// Mitsubishi GX Developer project: PLC_PCO520L2   PLC: Q06UDEH   Autoclave Auto Flow

PROGRAM AT_AC
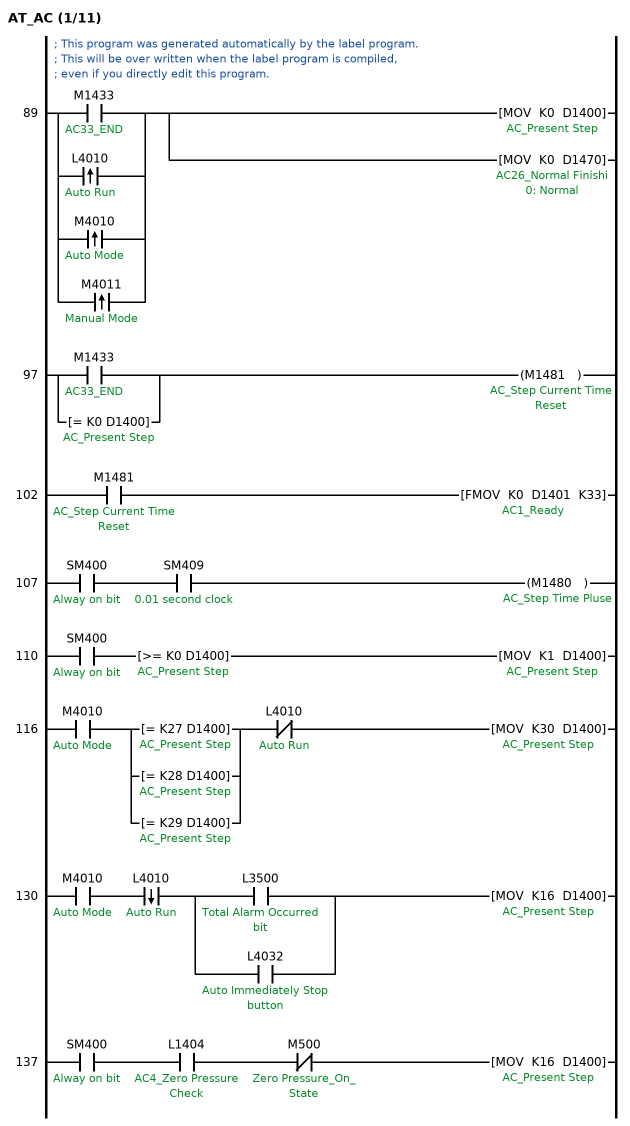
; This program was generated automatically by the label program.
; This will be over written when the label program is compiled,
; even if you directly edit this program.
89    LD      M1433  ; AC33_END
      ORP     L4010  ; Auto Run
      ORP     M4010  ; Auto Mode
      ORP     M4011  ; Manual Mode
      MOV     K0 D1400  ; AC_Present Step
      MOV     K0 D1470  ; AC26_Normal Finishi 0: Normal
97    LD      M1433  ; AC33_END
      OR=     K0 D1400  ; AC_Present Step
      OUT     M1481  ; AC_Step Current Time Reset
102   LD      M1481  ; AC_Step Current Time Reset
      FMOV    K0 D1401 K33  ; AC1_Ready
107   LD      SM400  ; Alway on bit
      AND     SM409  ; 0.01 second clock
      OUT     M1480  ; AC_Step Time Pluse
110   LD      SM400  ; Alway on bit
      AND>=   K0 D1400  ; AC_Present Step
      MOV     K1 D1400
116   LD      M4010  ; Auto Mode
      LD=     K27 D1400  ; AC_Present Step
      OR=     K28 D1400  ; AC_Present Step
      OR=     K29 D1400  ; AC_Present Step
      ANB
      ANI     L4010  ; Auto Run
      MOV     K30 D1400
130   LD      M4010  ; Auto Mode
      ANDF    L4010  ; Auto Run
      LD      L3500  ; Total Alarm Occurred bit
      OR      L4032  ; Auto Immediately Stop button
      ANB
      MOV     K16 D1400
137   LD      SM400  ; Alway on bit
      AND     L1404  ; AC4_Zero Pressure Check
      ANI     M500  ; Zero Pressure_On_State
      MOV     K16 D1400
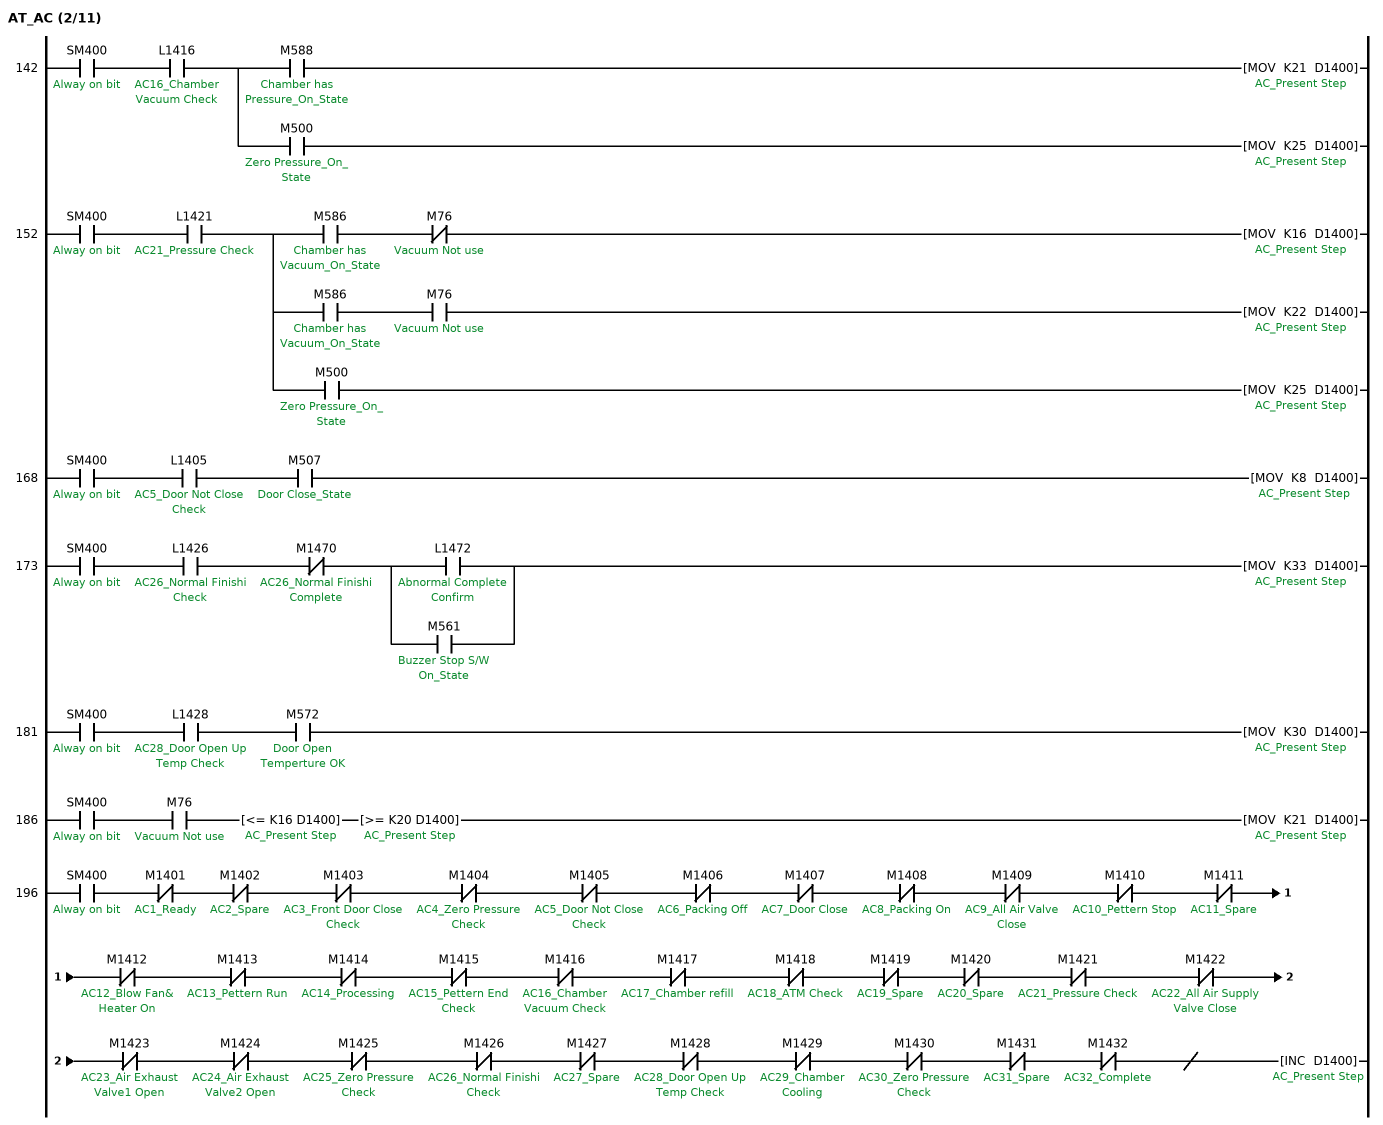
142   LD      SM400  ; Alway on bit
      AND     L1416  ; AC16_Chamber Vacuum Check
      MPS
      AND     M588  ; Chamber has Pressure_On_State
      MOV     K21 D1400
      MPP
      AND     M500  ; Zero Pressure_On_State
      MOV     K25 D1400
152   LD      SM400  ; Alway on bit
      AND     L1421  ; AC21_Pressure Check
      MPS
      AND     M586  ; Chamber has Vacuum_On_State
      ANI     M76  ; Vacuum Not use
      MOV     K16 D1400
      MRD
      AND     M586  ; Chamber has Vacuum_On_State
      AND     M76  ; Vacuum Not use
      MOV     K22 D1400
      MPP
      AND     M500  ; Zero Pressure_On_State
      MOV     K25 D1400
168   LD      SM400  ; Alway on bit
      AND     L1405  ; AC5_Door Not Close Check
      AND     M507  ; Door Close_State
      MOV     K8 D1400
173   LD      SM400  ; Alway on bit
      AND     L1426  ; AC26_Normal Finishi Check
      ANI     M1470  ; AC26_Normal Finishi Complete
      LD      L1472  ; Abnormal Complete Confirm
      OR      M561  ; Buzzer Stop S/W On_State
      ANB
      MOV     K33 D1400
181   LD      SM400  ; Alway on bit
      AND     L1428  ; AC28_Door Open Up Temp Check
      AND     M572  ; Door Open Temperture OK
      MOV     K30 D1400
186   LD      SM400  ; Alway on bit
      AND     M76  ; Vacuum Not use
      AND<=   K16 D1400  ; AC_Present Step
      AND>=   K20 D1400  ; AC_Present Step
      MOV     K21 D1400
196   LD      SM400  ; Alway on bit
      ANI     M1401  ; AC1_Ready
      ANI     M1402  ; AC2_Spare
      ANI     M1403  ; AC3_Front Door Close Check
      ANI     M1404  ; AC4_Zero Pressure Check
      ANI     M1405  ; AC5_Door Not Close Check
      ANI     M1406  ; AC6_Packing Off
      ANI     M1407  ; AC7_Door Close
      ANI     M1408  ; AC8_Packing On
      ANI     M1409  ; AC9_All Air Valve Close
      ANI     M1410  ; AC10_Pettern Stop
      ANI     M1411  ; AC11_Spare
      ANI     M1412  ; AC12_Blow Fan& Heater On
      ANI     M1413  ; AC13_Pettern Run
      ANI     M1414  ; AC14_Processing
      ANI     M1415  ; AC15_Pettern End Check
      ANI     M1416  ; AC16_Chamber Vacuum Check
      ANI     M1417  ; AC17_Chamber refill
      ANI     M1418  ; AC18_ATM Check
      ANI     M1419  ; AC19_Spare
      ANI     M1420  ; AC20_Spare
      ANI     M1421  ; AC21_Pressure Check
      ANI     M1422  ; AC22_All Air Supply Valve Close
      ANI     M1423  ; AC23_Air Exhaust Valve1 Open
      ANI     M1424  ; AC24_Air Exhaust Valve2 Open
      ANI     M1425  ; AC25_Zero Pressure Check
      ANI     M1426  ; AC26_Normal Finishi Check
      ANI     M1427  ; AC27_Spare
      ANI     M1428  ; AC28_Door Open Up Temp Check
      ANI     M1429  ; AC29_Chamber Cooling
      ANI     M1430  ; AC30_Zero Pressure Check
      ANI     M1431  ; AC31_Spare
      ANI     M1432  ; AC32_Complete
      INV
      INC     D1400
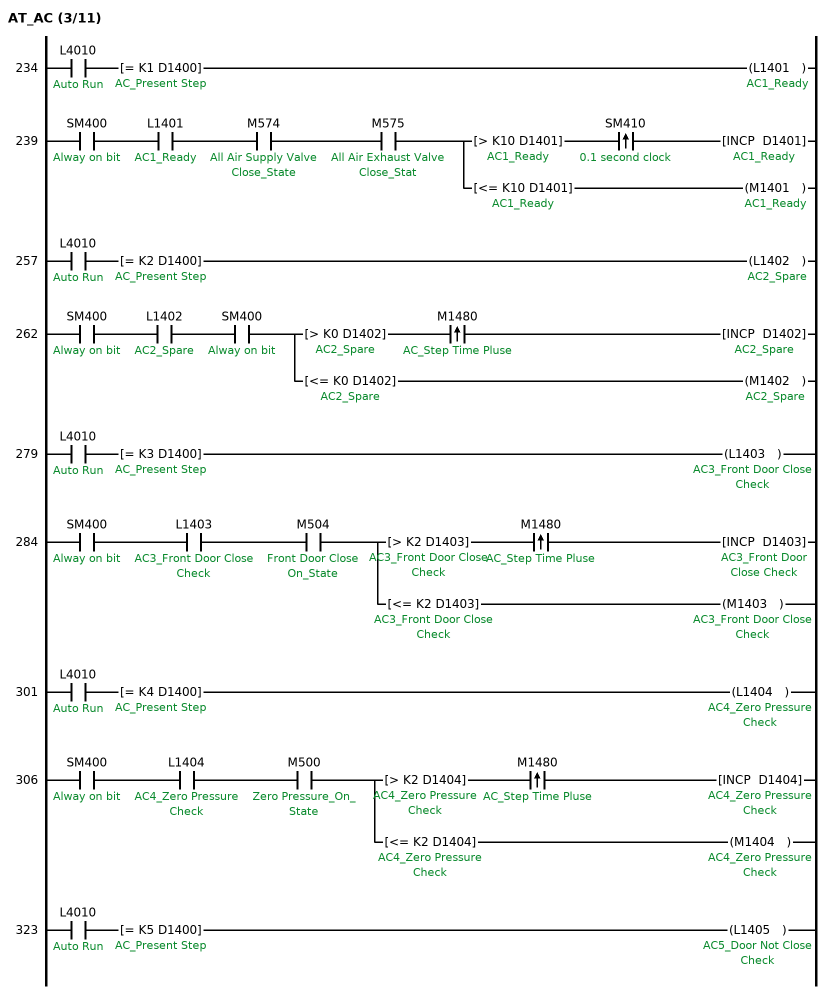
; 
234   LD      L4010  ; Auto Run
      AND=    K1 D1400  ; AC_Present Step
      OUT     L1401  ; AC1_Ready
239   LD      SM400  ; Alway on bit
      AND     L1401  ; AC1_Ready
      AND     M574  ; All Air Supply Valve Close_State
      AND     M575  ; All Air Exhaust Valve Close_Stat
      MPS
      AND>    K10 D1401  ; AC1_Ready
      ANDP    SM410  ; 0.1 second clock
      INCP    D1401
      MPP
      AND<=   K10 D1401  ; AC1_Ready
      OUT     M1401  ; AC1_Ready
; 
257   LD      L4010  ; Auto Run
      AND=    K2 D1400  ; AC_Present Step
      OUT     L1402  ; AC2_Spare
262   LD      SM400  ; Alway on bit
      AND     L1402  ; AC2_Spare
      AND     SM400  ; Alway on bit
      MPS
      AND>    K0 D1402  ; AC2_Spare
      ANDP    M1480  ; AC_Step Time Pluse
      INCP    D1402
      MPP
      AND<=   K0 D1402  ; AC2_Spare
      OUT     M1402  ; AC2_Spare
; 
279   LD      L4010  ; Auto Run
      AND=    K3 D1400  ; AC_Present Step
      OUT     L1403  ; AC3_Front Door Close Check
284   LD      SM400  ; Alway on bit
      AND     L1403  ; AC3_Front Door Close Check
      AND     M504  ; Front Door Close On_State
      MPS
      AND>    K2 D1403  ; AC3_Front Door Close Check
      ANDP    M1480  ; AC_Step Time Pluse
      INCP    D1403
      MPP
      AND<=   K2 D1403  ; AC3_Front Door Close Check
      OUT     M1403  ; AC3_Front Door Close Check
; 
301   LD      L4010  ; Auto Run
      AND=    K4 D1400  ; AC_Present Step
      OUT     L1404  ; AC4_Zero Pressure Check
306   LD      SM400  ; Alway on bit
      AND     L1404  ; AC4_Zero Pressure Check
      AND     M500  ; Zero Pressure_On_State
      MPS
      AND>    K2 D1404  ; AC4_Zero Pressure Check
      ANDP    M1480  ; AC_Step Time Pluse
      INCP    D1404
      MPP
      AND<=   K2 D1404  ; AC4_Zero Pressure Check
      OUT     M1404  ; AC4_Zero Pressure Check
; 
323   LD      L4010  ; Auto Run
      AND=    K5 D1400  ; AC_Present Step
      OUT     L1405  ; AC5_Door Not Close Check
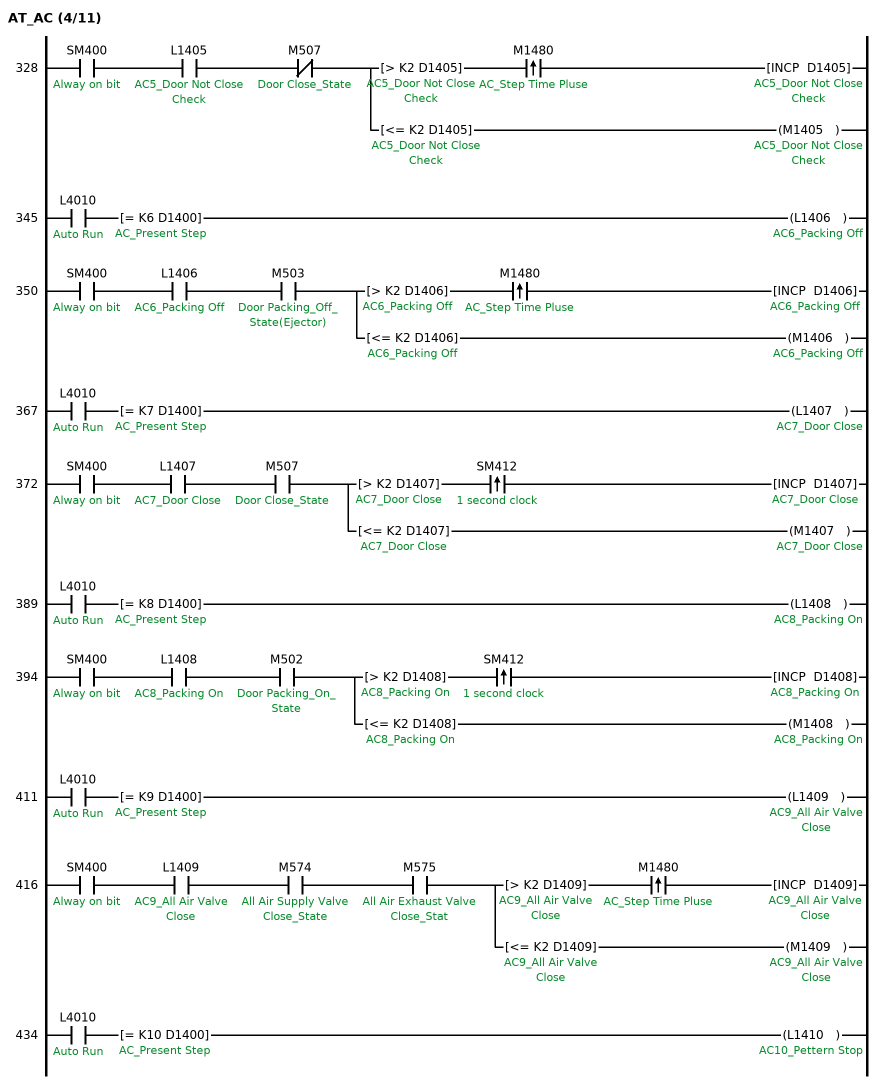
328   LD      SM400  ; Alway on bit
      AND     L1405  ; AC5_Door Not Close Check
      ANI     M507  ; Door Close_State
      MPS
      AND>    K2 D1405  ; AC5_Door Not Close Check
      ANDP    M1480  ; AC_Step Time Pluse
      INCP    D1405
      MPP
      AND<=   K2 D1405  ; AC5_Door Not Close Check
      OUT     M1405  ; AC5_Door Not Close Check
; 
345   LD      L4010  ; Auto Run
      AND=    K6 D1400  ; AC_Present Step
      OUT     L1406  ; AC6_Packing Off
350   LD      SM400  ; Alway on bit
      AND     L1406  ; AC6_Packing Off
      AND     M503  ; Door Packing_Off_State(Ejector)
      MPS
      AND>    K2 D1406  ; AC6_Packing Off
      ANDP    M1480  ; AC_Step Time Pluse
      INCP    D1406
      MPP
      AND<=   K2 D1406  ; AC6_Packing Off
      OUT     M1406  ; AC6_Packing Off
; 
367   LD      L4010  ; Auto Run
      AND=    K7 D1400  ; AC_Present Step
      OUT     L1407  ; AC7_Door Close
372   LD      SM400  ; Alway on bit
      AND     L1407  ; AC7_Door Close
      AND     M507  ; Door Close_State
      MPS
      AND>    K2 D1407  ; AC7_Door Close
      ANDP    SM412  ; 1 second clock
      INCP    D1407
      MPP
      AND<=   K2 D1407  ; AC7_Door Close
      OUT     M1407  ; AC7_Door Close
; 
389   LD      L4010  ; Auto Run
      AND=    K8 D1400  ; AC_Present Step
      OUT     L1408  ; AC8_Packing On
394   LD      SM400  ; Alway on bit
      AND     L1408  ; AC8_Packing On
      AND     M502  ; Door Packing_On_State
      MPS
      AND>    K2 D1408  ; AC8_Packing On
      ANDP    SM412  ; 1 second clock
      INCP    D1408
      MPP
      AND<=   K2 D1408  ; AC8_Packing On
      OUT     M1408  ; AC8_Packing On
; 
411   LD      L4010  ; Auto Run
      AND=    K9 D1400  ; AC_Present Step
      OUT     L1409  ; AC9_All Air Valve Close
416   LD      SM400  ; Alway on bit
      AND     L1409  ; AC9_All Air Valve Close
      AND     M574  ; All Air Supply Valve Close_State
      AND     M575  ; All Air Exhaust Valve Close_Stat
      MPS
      AND>    K2 D1409  ; AC9_All Air Valve Close
      ANDP    M1480  ; AC_Step Time Pluse
      INCP    D1409
      MPP
      AND<=   K2 D1409  ; AC9_All Air Valve Close
      OUT     M1409  ; AC9_All Air Valve Close
; 
434   LD      L4010  ; Auto Run
      AND=    K10 D1400  ; AC_Present Step
      OUT     L1410  ; AC10_Pettern Stop
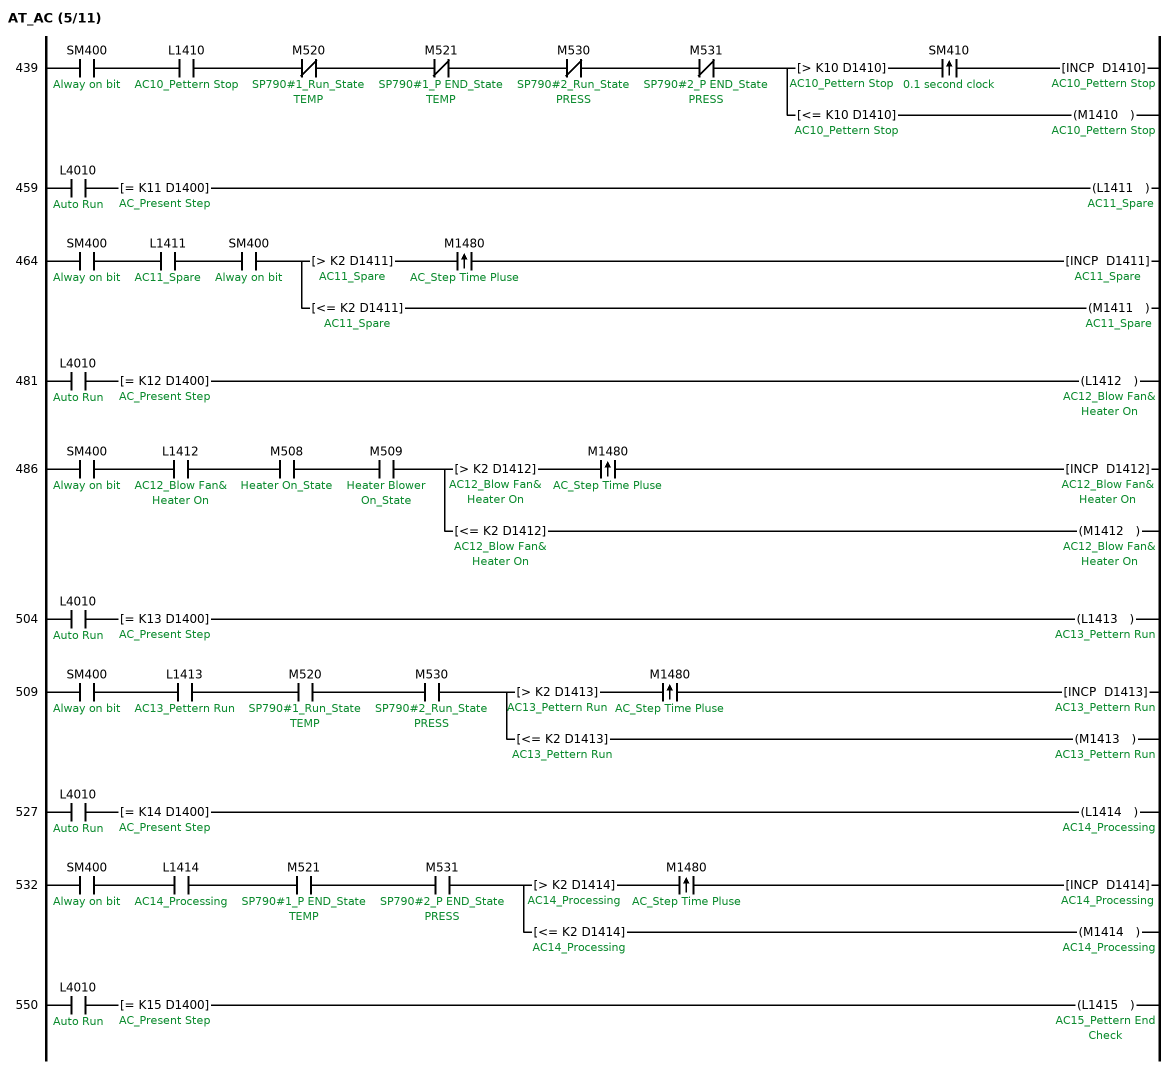
439   LD      SM400  ; Alway on bit
      AND     L1410  ; AC10_Pettern Stop
      ANI     M520  ; SP790#1_Run_State TEMP
      ANI     M521  ; SP790#1_P END_State TEMP
      ANI     M530  ; SP790#2_Run_State PRESS
      ANI     M531  ; SP790#2_P END_State PRESS
      MPS
      AND>    K10 D1410  ; AC10_Pettern Stop
      ANDP    SM410  ; 0.1 second clock
      INCP    D1410
      MPP
      AND<=   K10 D1410  ; AC10_Pettern Stop
      OUT     M1410  ; AC10_Pettern Stop
; 
459   LD      L4010  ; Auto Run
      AND=    K11 D1400  ; AC_Present Step
      OUT     L1411  ; AC11_Spare
464   LD      SM400  ; Alway on bit
      AND     L1411  ; AC11_Spare
      AND     SM400  ; Alway on bit
      MPS
      AND>    K2 D1411  ; AC11_Spare
      ANDP    M1480  ; AC_Step Time Pluse
      INCP    D1411
      MPP
      AND<=   K2 D1411  ; AC11_Spare
      OUT     M1411  ; AC11_Spare
; 
481   LD      L4010  ; Auto Run
      AND=    K12 D1400  ; AC_Present Step
      OUT     L1412  ; AC12_Blow Fan& Heater On
486   LD      SM400  ; Alway on bit
      AND     L1412  ; AC12_Blow Fan& Heater On
      AND     M508  ; Heater On_State
      AND     M509  ; Heater Blower On_State
      MPS
      AND>    K2 D1412  ; AC12_Blow Fan& Heater On
      ANDP    M1480  ; AC_Step Time Pluse
      INCP    D1412
      MPP
      AND<=   K2 D1412  ; AC12_Blow Fan& Heater On
      OUT     M1412  ; AC12_Blow Fan& Heater On
; 
504   LD      L4010  ; Auto Run
      AND=    K13 D1400  ; AC_Present Step
      OUT     L1413  ; AC13_Pettern Run
509   LD      SM400  ; Alway on bit
      AND     L1413  ; AC13_Pettern Run
      AND     M520  ; SP790#1_Run_State TEMP
      AND     M530  ; SP790#2_Run_State PRESS
      MPS
      AND>    K2 D1413  ; AC13_Pettern Run
      ANDP    M1480  ; AC_Step Time Pluse
      INCP    D1413
      MPP
      AND<=   K2 D1413  ; AC13_Pettern Run
      OUT     M1413  ; AC13_Pettern Run
; 
527   LD      L4010  ; Auto Run
      AND=    K14 D1400  ; AC_Present Step
      OUT     L1414  ; AC14_Processing
532   LD      SM400  ; Alway on bit
      AND     L1414  ; AC14_Processing
      AND     M521  ; SP790#1_P END_State TEMP
      AND     M531  ; SP790#2_P END_State PRESS
      MPS
      AND>    K2 D1414  ; AC14_Processing
      ANDP    M1480  ; AC_Step Time Pluse
      INCP    D1414
      MPP
      AND<=   K2 D1414  ; AC14_Processing
      OUT     M1414  ; AC14_Processing
; 
550   LD      L4010  ; Auto Run
      AND=    K15 D1400  ; AC_Present Step
      OUT     L1415  ; AC15_Pettern End Check
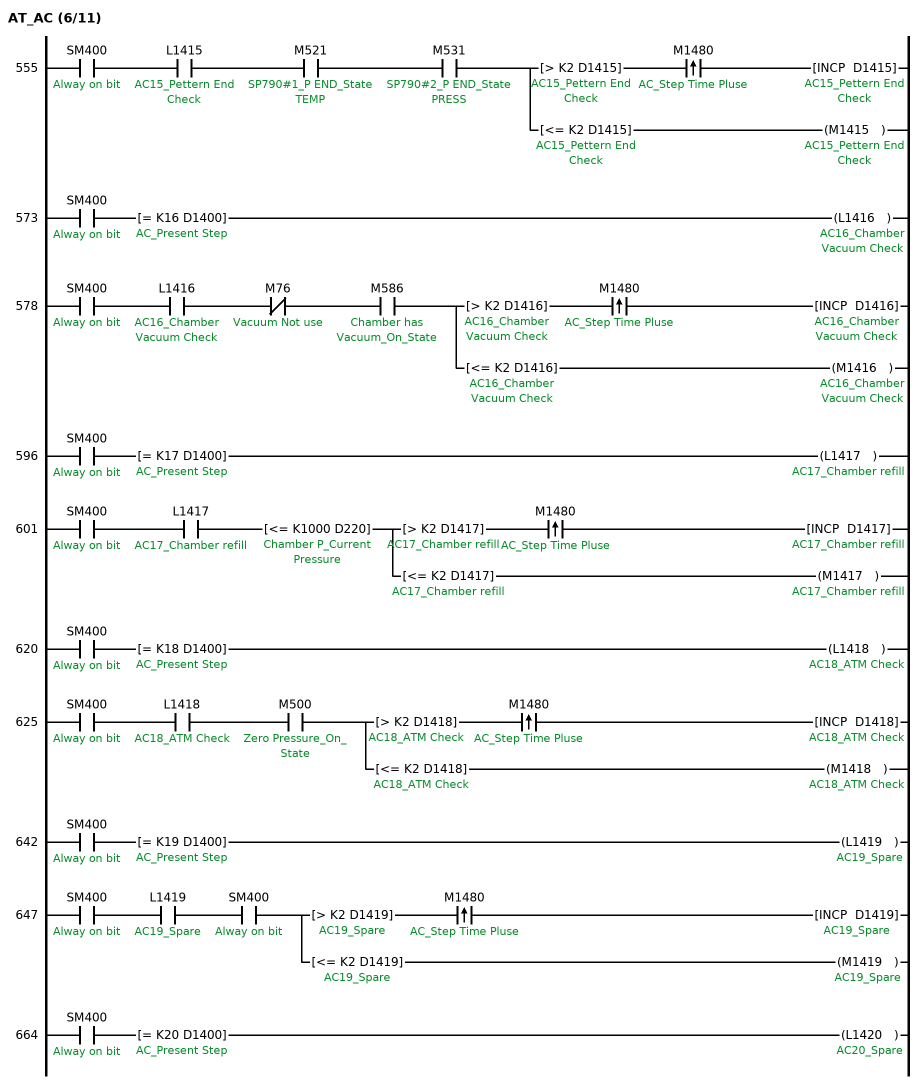
555   LD      SM400  ; Alway on bit
      AND     L1415  ; AC15_Pettern End Check
      AND     M521  ; SP790#1_P END_State TEMP
      AND     M531  ; SP790#2_P END_State PRESS
      MPS
      AND>    K2 D1415  ; AC15_Pettern End Check
      ANDP    M1480  ; AC_Step Time Pluse
      INCP    D1415
      MPP
      AND<=   K2 D1415  ; AC15_Pettern End Check
      OUT     M1415  ; AC15_Pettern End Check
; 
573   LD      SM400  ; Alway on bit
      AND=    K16 D1400  ; AC_Present Step
      OUT     L1416  ; AC16_Chamber Vacuum Check
578   LD      SM400  ; Alway on bit
      AND     L1416  ; AC16_Chamber Vacuum Check
      ANI     M76  ; Vacuum Not use
      AND     M586  ; Chamber has Vacuum_On_State
      MPS
      AND>    K2 D1416  ; AC16_Chamber Vacuum Check
      ANDP    M1480  ; AC_Step Time Pluse
      INCP    D1416
      MPP
      AND<=   K2 D1416  ; AC16_Chamber Vacuum Check
      OUT     M1416  ; AC16_Chamber Vacuum Check
; 
596   LD      SM400  ; Alway on bit
      AND=    K17 D1400  ; AC_Present Step
      OUT     L1417  ; AC17_Chamber refill
601   LD      SM400  ; Alway on bit
      AND     L1417  ; AC17_Chamber refill
      AND<=   K1000 D220  ; Chamber P_Current Pressure
      MPS
      AND>    K2 D1417  ; AC17_Chamber refill
      ANDP    M1480  ; AC_Step Time Pluse
      INCP    D1417
      MPP
      AND<=   K2 D1417  ; AC17_Chamber refill
      OUT     M1417  ; AC17_Chamber refill
; 
620   LD      SM400  ; Alway on bit
      AND=    K18 D1400  ; AC_Present Step
      OUT     L1418  ; AC18_ATM Check
625   LD      SM400  ; Alway on bit
      AND     L1418  ; AC18_ATM Check
      AND     M500  ; Zero Pressure_On_State
      MPS
      AND>    K2 D1418  ; AC18_ATM Check
      ANDP    M1480  ; AC_Step Time Pluse
      INCP    D1418
      MPP
      AND<=   K2 D1418  ; AC18_ATM Check
      OUT     M1418  ; AC18_ATM Check
; 
642   LD      SM400  ; Alway on bit
      AND=    K19 D1400  ; AC_Present Step
      OUT     L1419  ; AC19_Spare
647   LD      SM400  ; Alway on bit
      AND     L1419  ; AC19_Spare
      AND     SM400  ; Alway on bit
      MPS
      AND>    K2 D1419  ; AC19_Spare
      ANDP    M1480  ; AC_Step Time Pluse
      INCP    D1419
      MPP
      AND<=   K2 D1419  ; AC19_Spare
      OUT     M1419  ; AC19_Spare
; 
664   LD      SM400  ; Alway on bit
      AND=    K20 D1400  ; AC_Present Step
      OUT     L1420  ; AC20_Spare
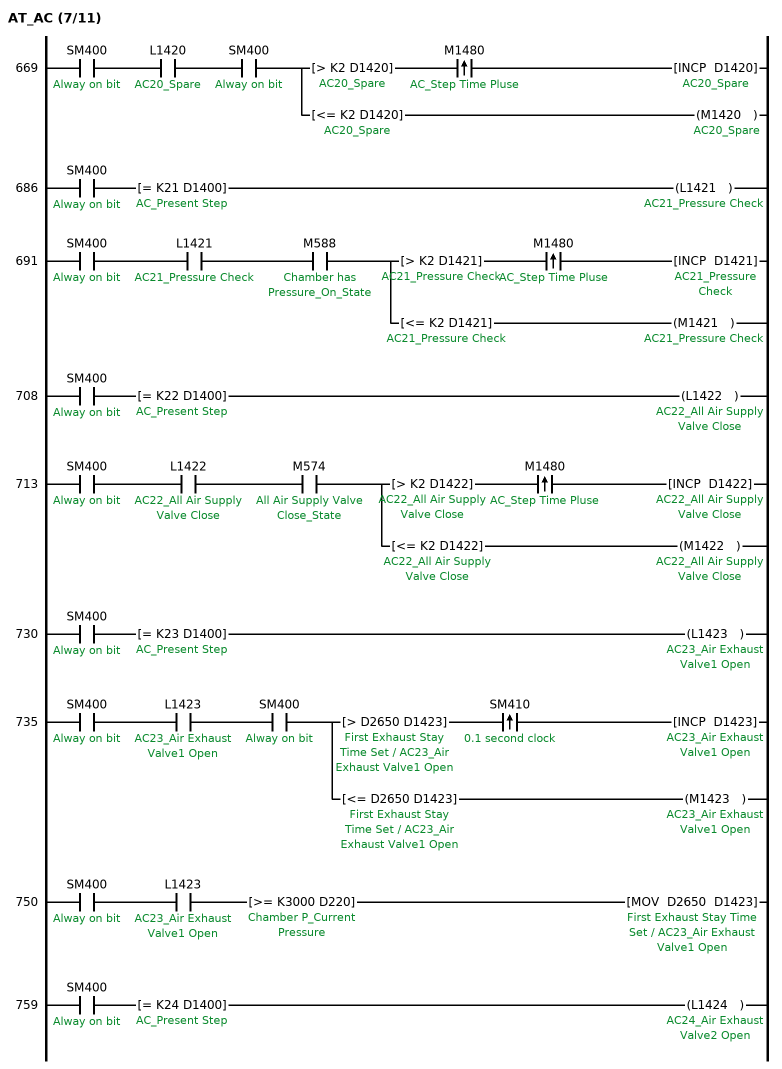
669   LD      SM400  ; Alway on bit
      AND     L1420  ; AC20_Spare
      AND     SM400  ; Alway on bit
      MPS
      AND>    K2 D1420  ; AC20_Spare
      ANDP    M1480  ; AC_Step Time Pluse
      INCP    D1420
      MPP
      AND<=   K2 D1420  ; AC20_Spare
      OUT     M1420  ; AC20_Spare
; 
686   LD      SM400  ; Alway on bit
      AND=    K21 D1400  ; AC_Present Step
      OUT     L1421  ; AC21_Pressure Check
691   LD      SM400  ; Alway on bit
      AND     L1421  ; AC21_Pressure Check
      AND     M588  ; Chamber has Pressure_On_State
      MPS
      AND>    K2 D1421  ; AC21_Pressure Check
      ANDP    M1480  ; AC_Step Time Pluse
      INCP    D1421
      MPP
      AND<=   K2 D1421  ; AC21_Pressure Check
      OUT     M1421  ; AC21_Pressure Check
; 
708   LD      SM400  ; Alway on bit
      AND=    K22 D1400  ; AC_Present Step
      OUT     L1422  ; AC22_All Air Supply Valve Close
713   LD      SM400  ; Alway on bit
      AND     L1422  ; AC22_All Air Supply Valve Close
      AND     M574  ; All Air Supply Valve Close_State
      MPS
      AND>    K2 D1422  ; AC22_All Air Supply Valve Close
      ANDP    M1480  ; AC_Step Time Pluse
      INCP    D1422
      MPP
      AND<=   K2 D1422  ; AC22_All Air Supply Valve Close
      OUT     M1422  ; AC22_All Air Supply Valve Close
; 
730   LD      SM400  ; Alway on bit
      AND=    K23 D1400  ; AC_Present Step
      OUT     L1423  ; AC23_Air Exhaust Valve1 Open
735   LD      SM400  ; Alway on bit
      AND     L1423  ; AC23_Air Exhaust Valve1 Open
      AND     SM400  ; Alway on bit
      MPS
      AND>    D2650 D1423  ; First Exhaust Stay Time Set / AC23_Air Exhaust Valve1 Open
      ANDP    SM410  ; 0.1 second clock
      INCP    D1423
      MPP
      AND<=   D2650 D1423  ; First Exhaust Stay Time Set / AC23_Air Exhaust Valve1 Open
      OUT     M1423  ; AC23_Air Exhaust Valve1 Open
750   LD      SM400  ; Alway on bit
      AND     L1423  ; AC23_Air Exhaust Valve1 Open
      AND>=   K3000 D220  ; Chamber P_Current Pressure
      MOV     D2650 D1423
; 
759   LD      SM400  ; Alway on bit
      AND=    K24 D1400  ; AC_Present Step
      OUT     L1424  ; AC24_Air Exhaust Valve2 Open
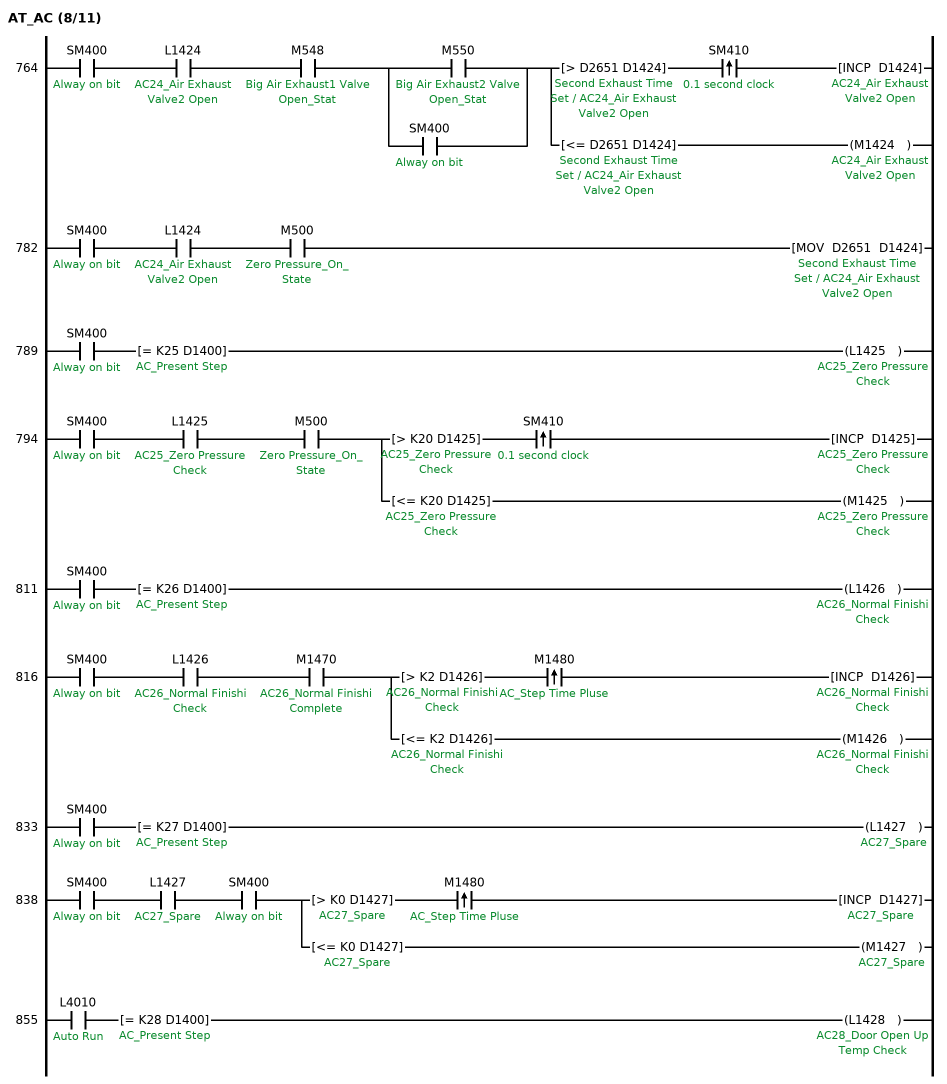
764   LD      SM400  ; Alway on bit
      AND     L1424  ; AC24_Air Exhaust Valve2 Open
      AND     M548  ; Big Air Exhaust1 Valve Open_Stat
      LD      M550  ; Big Air Exhaust2 Valve Open_Stat
      OR      SM400  ; Alway on bit
      ANB
      MPS
      AND>    D2651 D1424  ; Second Exhaust Time Set / AC24_Air Exhaust Valve2 Open
      ANDP    SM410  ; 0.1 second clock
      INCP    D1424
      MPP
      AND<=   D2651 D1424  ; Second Exhaust Time Set / AC24_Air Exhaust Valve2 Open
      OUT     M1424  ; AC24_Air Exhaust Valve2 Open
782   LD      SM400  ; Alway on bit
      AND     L1424  ; AC24_Air Exhaust Valve2 Open
      AND     M500  ; Zero Pressure_On_State
      MOV     D2651 D1424
; 
789   LD      SM400  ; Alway on bit
      AND=    K25 D1400  ; AC_Present Step
      OUT     L1425  ; AC25_Zero Pressure Check
794   LD      SM400  ; Alway on bit
      AND     L1425  ; AC25_Zero Pressure Check
      AND     M500  ; Zero Pressure_On_State
      MPS
      AND>    K20 D1425  ; AC25_Zero Pressure Check
      ANDP    SM410  ; 0.1 second clock
      INCP    D1425
      MPP
      AND<=   K20 D1425  ; AC25_Zero Pressure Check
      OUT     M1425  ; AC25_Zero Pressure Check
; 
811   LD      SM400  ; Alway on bit
      AND=    K26 D1400  ; AC_Present Step
      OUT     L1426  ; AC26_Normal Finishi Check
816   LD      SM400  ; Alway on bit
      AND     L1426  ; AC26_Normal Finishi Check
      AND     M1470  ; AC26_Normal Finishi Complete
      MPS
      AND>    K2 D1426  ; AC26_Normal Finishi Check
      ANDP    M1480  ; AC_Step Time Pluse
      INCP    D1426
      MPP
      AND<=   K2 D1426  ; AC26_Normal Finishi Check
      OUT     M1426  ; AC26_Normal Finishi Check
; 
833   LD      SM400  ; Alway on bit
      AND=    K27 D1400  ; AC_Present Step
      OUT     L1427  ; AC27_Spare
838   LD      SM400  ; Alway on bit
      AND     L1427  ; AC27_Spare
      AND     SM400  ; Alway on bit
      MPS
      AND>    K0 D1427  ; AC27_Spare
      ANDP    M1480  ; AC_Step Time Pluse
      INCP    D1427
      MPP
      AND<=   K0 D1427  ; AC27_Spare
      OUT     M1427  ; AC27_Spare
; 
855   LD      L4010  ; Auto Run
      AND=    K28 D1400  ; AC_Present Step
      OUT     L1428  ; AC28_Door Open Up Temp Check
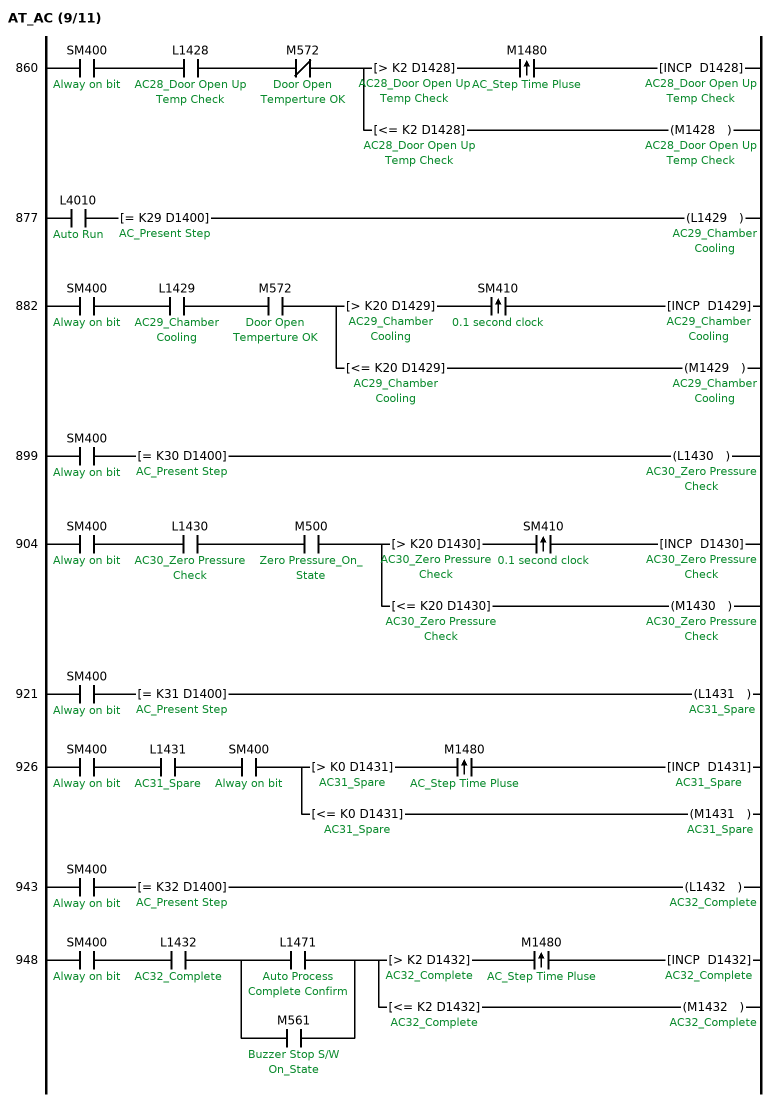
860   LD      SM400  ; Alway on bit
      AND     L1428  ; AC28_Door Open Up Temp Check
      ANI     M572  ; Door Open Temperture OK
      MPS
      AND>    K2 D1428  ; AC28_Door Open Up Temp Check
      ANDP    M1480  ; AC_Step Time Pluse
      INCP    D1428
      MPP
      AND<=   K2 D1428  ; AC28_Door Open Up Temp Check
      OUT     M1428  ; AC28_Door Open Up Temp Check
; 
877   LD      L4010  ; Auto Run
      AND=    K29 D1400  ; AC_Present Step
      OUT     L1429  ; AC29_Chamber Cooling
882   LD      SM400  ; Alway on bit
      AND     L1429  ; AC29_Chamber Cooling
      AND     M572  ; Door Open Temperture OK
      MPS
      AND>    K20 D1429  ; AC29_Chamber Cooling
      ANDP    SM410  ; 0.1 second clock
      INCP    D1429
      MPP
      AND<=   K20 D1429  ; AC29_Chamber Cooling
      OUT     M1429  ; AC29_Chamber Cooling
; 
899   LD      SM400  ; Alway on bit
      AND=    K30 D1400  ; AC_Present Step
      OUT     L1430  ; AC30_Zero Pressure Check
904   LD      SM400  ; Alway on bit
      AND     L1430  ; AC30_Zero Pressure Check
      AND     M500  ; Zero Pressure_On_State
      MPS
      AND>    K20 D1430  ; AC30_Zero Pressure Check
      ANDP    SM410  ; 0.1 second clock
      INCP    D1430
      MPP
      AND<=   K20 D1430  ; AC30_Zero Pressure Check
      OUT     M1430  ; AC30_Zero Pressure Check
; 
921   LD      SM400  ; Alway on bit
      AND=    K31 D1400  ; AC_Present Step
      OUT     L1431  ; AC31_Spare
926   LD      SM400  ; Alway on bit
      AND     L1431  ; AC31_Spare
      AND     SM400  ; Alway on bit
      MPS
      AND>    K0 D1431  ; AC31_Spare
      ANDP    M1480  ; AC_Step Time Pluse
      INCP    D1431
      MPP
      AND<=   K0 D1431  ; AC31_Spare
      OUT     M1431  ; AC31_Spare
; 
943   LD      SM400  ; Alway on bit
      AND=    K32 D1400  ; AC_Present Step
      OUT     L1432  ; AC32_Complete
948   LD      SM400  ; Alway on bit
      AND     L1432  ; AC32_Complete
      LD      L1471  ; Auto Process Complete Confirm
      OR      M561  ; Buzzer Stop S/W On_State
      ANB
      MPS
      AND>    K2 D1432  ; AC32_Complete
      ANDP    M1480  ; AC_Step Time Pluse
      INCP    D1432
      MPP
      AND<=   K2 D1432  ; AC32_Complete
      OUT     M1432  ; AC32_Complete
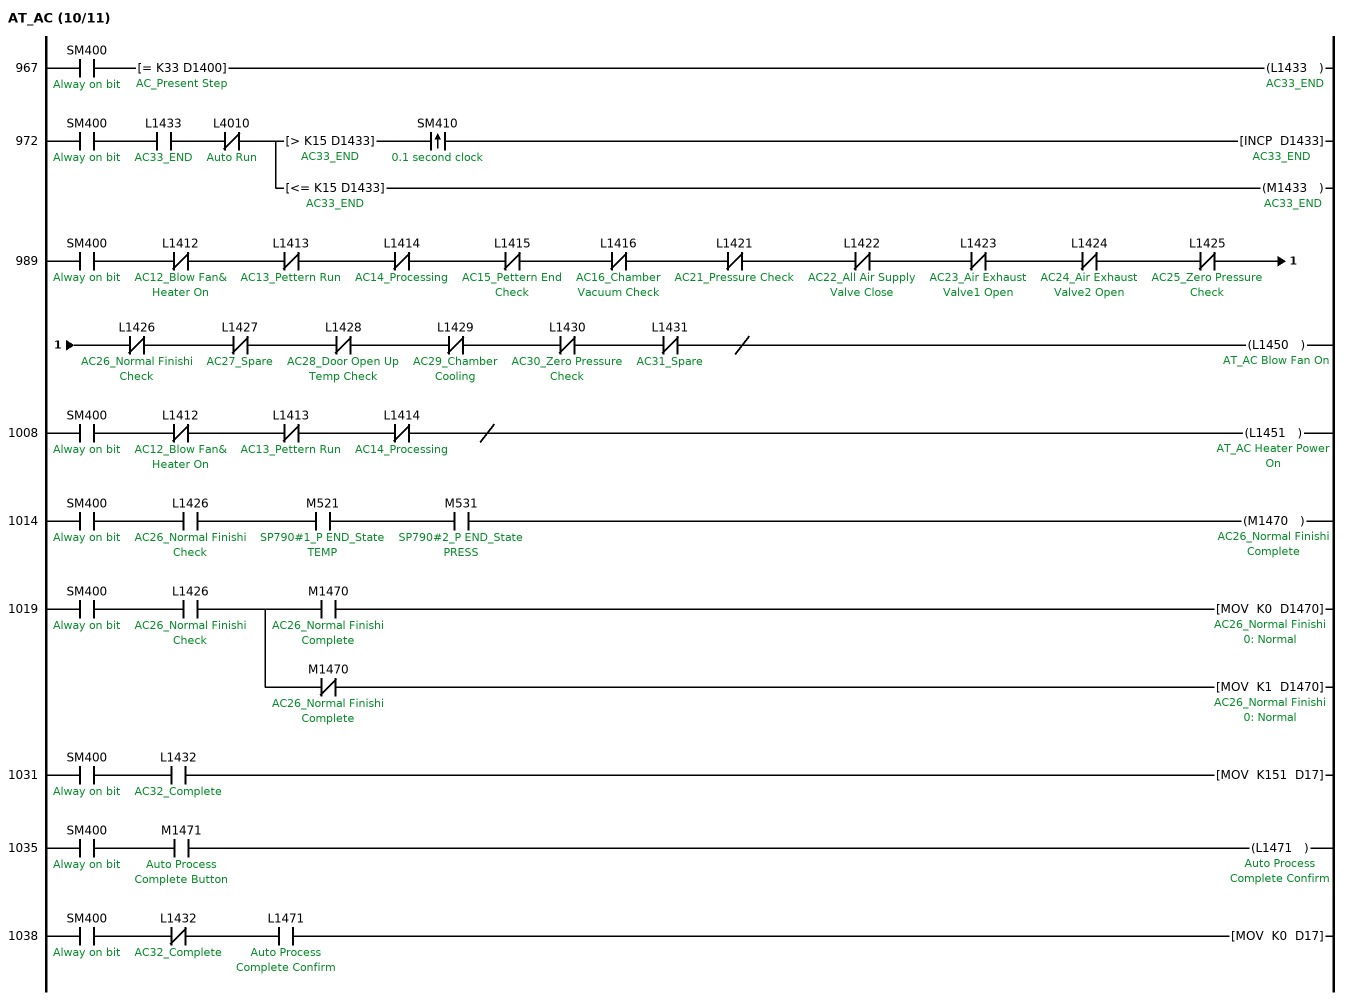
; 
967   LD      SM400  ; Alway on bit
      AND=    K33 D1400  ; AC_Present Step
      OUT     L1433  ; AC33_END
972   LD      SM400  ; Alway on bit
      AND     L1433  ; AC33_END
      ANI     L4010  ; Auto Run
      MPS
      AND>    K15 D1433  ; AC33_END
      ANDP    SM410  ; 0.1 second clock
      INCP    D1433
      MPP
      AND<=   K15 D1433  ; AC33_END
      OUT     M1433  ; AC33_END
; 
989   LD      SM400  ; Alway on bit
      ANI     L1412  ; AC12_Blow Fan& Heater On
      ANI     L1413  ; AC13_Pettern Run
      ANI     L1414  ; AC14_Processing
      ANI     L1415  ; AC15_Pettern End Check
      ANI     L1416  ; AC16_Chamber Vacuum Check
      ANI     L1421  ; AC21_Pressure Check
      ANI     L1422  ; AC22_All Air Supply Valve Close
      ANI     L1423  ; AC23_Air Exhaust Valve1 Open
      ANI     L1424  ; AC24_Air Exhaust Valve2 Open
      ANI     L1425  ; AC25_Zero Pressure Check
      ANI     L1426  ; AC26_Normal Finishi Check
      ANI     L1427  ; AC27_Spare
      ANI     L1428  ; AC28_Door Open Up Temp Check
      ANI     L1429  ; AC29_Chamber Cooling
      ANI     L1430  ; AC30_Zero Pressure Check
      ANI     L1431  ; AC31_Spare
      INV
      OUT     L1450  ; AT_AC Blow Fan On
1008  LD      SM400  ; Alway on bit
      ANI     L1412  ; AC12_Blow Fan& Heater On
      ANI     L1413  ; AC13_Pettern Run
      ANI     L1414  ; AC14_Processing
      INV
      OUT     L1451  ; AT_AC Heater Power On
1014  LD      SM400  ; Alway on bit
      AND     L1426  ; AC26_Normal Finishi Check
      AND     M521  ; SP790#1_P END_State TEMP
      AND     M531  ; SP790#2_P END_State PRESS
      OUT     M1470  ; AC26_Normal Finishi Complete
1019  LD      SM400  ; Alway on bit
      AND     L1426  ; AC26_Normal Finishi Check
      MPS
      AND     M1470  ; AC26_Normal Finishi Complete
      MOV     K0 D1470
      MPP
      ANI     M1470  ; AC26_Normal Finishi Complete
      MOV     K1 D1470
; 
1031  LD      SM400  ; Alway on bit
      AND     L1432  ; AC32_Complete
      MOV     K151 D17
1035  LD      SM400  ; Alway on bit
      AND     M1471  ; Auto Process Complete Button
      OUT     L1471  ; Auto Process Complete Confirm
1038  LD      SM400  ; Alway on bit
      ANI     L1432  ; AC32_Complete
      AND     L1471  ; Auto Process Complete Confirm
      MOV     K0 D17
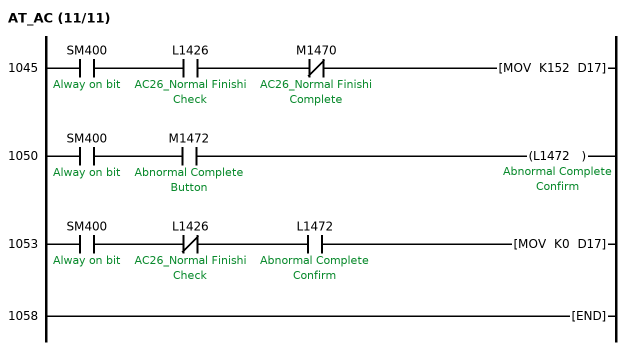
; 
1045  LD      SM400  ; Alway on bit
      AND     L1426  ; AC26_Normal Finishi Check
      ANI     M1470  ; AC26_Normal Finishi Complete
      MOV     K152 D17
1050  LD      SM400  ; Alway on bit
      AND     M1472  ; Abnormal Complete Button
      OUT     L1472  ; Abnormal Complete Confirm
1053  LD      SM400  ; Alway on bit
      ANI     L1426  ; AC26_Normal Finishi Check
      AND     L1472  ; Abnormal Complete Confirm
      MOV     K0 D17
1058  END
END_PROGRAM
